FUNCTION_BLOCK CiA_DS402Statusword_StaeubliCS8 EXTENDS CiA_DS402Statusword
VAR_INPUT
END_VAR
VAR_OUTPUT	
	FollowCmdValue			: bool;  //Bit 12: Drive follows command (CSP/CSV)
	FollowingError			: BOOL; // Bit 13: Following error occured
	Calibrated				: BOOL; // Bit 14: Motor calibrated
END_VAR

METHOD PUBLIC readStatusword : BOOL
VAR_INPUT
	Statusword 		:	UINT;

END_VAR
FollowCmdValue												:= Statusword.12 ;
FollowingError												:= Statusword.13 ;
Calibrated													:= Statusword.14 ;

readStatusword												:= SUPER^.readStatusword(Statusword);
END_METHOD

END_FUNCTION_BLOCK

(* stored: Version 1.1.0.1, ProductVersion 3.1.4024.13
   POU CiA_DS402Statusword_StaeubliCS8: Id {059bae0e-e4a8-4717-a4c9-962fb1dd2811}, SpecialFunc None
   Method readStatusword: Id {95b0b135-a7c4-4afe-9f0c-88a951cd1f2e} *)
